// TIA Portal V17 export
// export: Created 2025-03-07T09:19:56.0957426Z, ExportSetting WithDefaults, DisplayName Totally Integrated Automation Portal, DisplayVersion V17 Update 8, DisplayName TIA Portal Openness, DisplayVersion V17 Update 8, DisplayName TIA Portal Version Control Interface, DisplayVersion V17, DisplayName SINAMICS Startdrive Advanced, DisplayVersion V17 SP2, DisplayName SINAMICS Startdrive G110M, G120, G120C, G120D, G120P, G115D, DisplayVersion V17 SP2, DisplayName SINAMICS Startdrive G130, G150, S120, S150, SINAMICS MV, S210, DisplayVersion V17 SP2, DisplayName STEP 7 Professional, DisplayVersion V17 Update 8, DisplayName SINUMERIK ONE STEP 7 Toolbox, DisplayVersion V17 Update 12, DisplayName SINUMERIK 840D sl STEP 7 Toolbox, DisplayVersion V17 Update 12, DisplayName STEP 7 Safety, DisplayVersion V17 Update 6, DisplayName WinCC Advanced, DisplayVersion V17 Update 8
TYPE "LOAD_ROBOT"
// stored: IsFailsafeCompliant false
   STRUCT
      TO_FIXT : Struct
         PART_A_LOADED_FIXT1 : Bool;   // PART 1 LOADED ARM 1 / PART A LOADED FIXT 1
         PART_B_LOADED_FIXT1 : Bool;   // PART 2 LOADED ARM 1 / PART B LOADED FIXT 1
         PART_C_LOADED_FIXT1 : Bool;   // PART 3 LOADED ARM 1 / PART C LOADED FIXT 1
         PART_D_LOADED_FIXT1 : Bool;   // PART 4 LOADED ARM 1 / PART D LOADED FIXT 1
         PART_A_LOADED_FIXT2 : Bool;   // PART 1 LOADED ARM 2 / PART A LOADED FIXT 2
         PART_B_LOADED_FIXT2 : Bool;   // PART 2 LOADED ARM 2 / PART B LOADED FIXT 2
         PART_C_LOADED_FIXT2 : Bool;   // PART 3 LOADED ARM 2 / PART C LOADED FIXT 2
         PART_D_LOADED_FIXT2 : Bool;   // PART 4 LOADED ARM 2 / PART D LOADED FIXT 2
         PARTS_LOADED_FIXT1 : Bool;   // PARTS LOADED ARM 1 / PARTS LOADED FIXT 1
         PARTS_LOADED_FIXT2 : Bool;   // PARTS LOADED ARM 2 / PARTS LOADED FIXT 2
         I_PART_PRESENT_A : Bool;   // INPUT PART PRESENT A
         I_PART_PRESENT_B : Bool;   // INPUT PART PRESENT B
         I_PART_PRESENT_C : Bool;   // INPUT PART PRESENT C
         I_PART_PRESENT_D : Bool;   // INPUT PART PRESENT D
         PART_A_UNLOADED_FIXT1 : Bool;   // PART 1 UNLOADED ARM 1 / PART A UNLOADED FIXT 1
         PART_B_UNLOADED_FIXT1 : Bool;   // PART 2 UNLOADED ARM 1 / PART B UNLOADED FIXT 1
         PART_C_UNLOADED_FIXT1 : Bool;   // PART 3 UNLOADED ARM 1 / PART C UNLOADED FIXT 1
         PART_D_UNLOADED_FIXT1 : Bool;   // PART 4 UNLOADED ARM 1 / PART D UNLOADED FIXT 1
         PART_A_UNLOADED_FIXT2 : Bool;   // PART 1 UNLOADED ARM 2 / PART A UNLOADED FIXT 2
         PART_B_UNLOADED_FIXT2 : Bool;   // PART 2 UNLOADED ARM 2 / PART B UNLOADED FIXT 2
         PART_C_UNLOADED_FIXT2 : Bool;   // PART 3 UNLOADED ARM 2 / PART C UNLOADED FIXT 2
         PART_D_UNLOADED_FIXT2 : Bool;   // PART 4 UNLOADED ARM 2 / PART D UNLOADED FIXT 2
         PARTS_UNLOADED_FIXT1 : Bool;   // PARTS UNLOADED ARM 1 / PARTS UNLOADED FIXT 1
         PARTS_UNLOADED_FIXT2 : Bool;   // PARTS UNLOADED ARM 2 / PARTS UNLOADED FIXT 2
         AUX_PART_A_LOADED_FIXT1 : Bool;   // AUX PART A LOADED FIXT1
         AUX_PART_B_LOADED_FIXT1 : Bool;   // AUX PART B LOADED FIXT1
         AUX_PART_C_LOADED_FIXT1 : Bool;   // AUX PART C LOADED FIXT1
         AUX_PART_D_LOADED_FIXT1 : Bool;   // AUX PART D LOADED FIXT1
         AUX_PART_A_LOADED_FIXT2 : Bool;   // AUX PART A LOADED FIXT2
         AUX_PART_B_LOADED_FIXT2 : Bool;   // AUX PART B LOADED FIXT2
         AUX_PART_C_LOADED_FIXT2 : Bool;   // AUX PART C LOADED FIXT2
         AUX_PART_D_LOADED_FIXT2 : Bool;   // AUX PART D LOADED FIXT2
         NO_PARTS_AT_FIXT1 : Bool;   // NO PARTS AT ARM 1 / NO PARTS AT FIXT 1
         NO_PARTS_AT_FIXT2 : Bool;   // NO PARTS AT ARM 2 / NO PARTS AT FIXT 2
         PART_A_LOADED_FIXT1_P : Bool;   // PART 1 LOADED ARM 1 PULSE / PART A LOADED FIXT 1 PULSE
         PART_B_LOADED_FIXT1_P : Bool;   // PART 2 LOADED ARM 1 PULSE / PART B LOADED FIXT 1 PULSE
         PART_C_LOADED_FIXT1_P : Bool;   // PART 3 LOADED ARM 1 PULSE / PART C LOADED FIXT 1 PULSE
         PART_D_LOADED_FIXT1_P : Bool;   // PART 4 LOADED ARM 1 PULSE / PART D LOADED FIXT 1 PULSE
         PART_A_LOADED_FIXT2_P : Bool;   // PART 1 LOADED ARM 2 PULSE / PART A LOADED FIXT 2 PULSE
         PART_B_LOADED_FIXT2_P : Bool;   // PART 2 LOADED ARM 2 PULSE / PART B LOADED FIXT 2 PULSE
         PART_C_LOADED_FIXT2_P : Bool;   // PART 3 LOADED ARM 2 PULSE / PART C LOADED FIXT 2 PULSE
         PART_D_LOADED_FIXT2_P : Bool;   // PART 4 LOADED ARM 2 PULSE / PART D LOADED FIXT 2 PULSE
         PARTS_LOADED_FIXT1_P : Bool;   // PARTS LOADED ARM 1 PULSE / PARTS LOADED FIXT 1 PULSE
         PARTS_LOADED_FIXT2_P : Bool;   // PARTS LOADED ARM 2 PULSE / PARTS LOADED FIXT 2 PULSE
         ANY_PART_LOADED : Bool;   // ANY PART LOADED
         ANY_PART_UNLOADED : Bool;   // ANY PART UNLOADED
         ENABLE_LOAD_UNLOAD : Bool;   // ENABLE TO LOAD UNLOAD LOADER TO TRANSFER
         PARTS_LOADING : Bool;   // THE GANTRY IS LOADING PARTS
         PART_A_UNLOADED_FIXT1_P : Bool;   // PART 1 UNLOADED ARM 1 PULSE / PART A UNLOADED FIXT 1 PULSE
         PART_B_UNLOADED_FIXT1_P : Bool;   // PART 2 UNLOADED ARM 1 PULSE / PART B UNLOADED FIXT 1 PULSE
         PART_C_UNLOADED_FIXT1_P : Bool;   // PART 3 UNLOADED ARM 1 PULSE / PART C UNLOADED FIXT 1 PULSE
         PART_D_UNLOADED_FIXT1_P : Bool;   // PART 4 UNLOADED ARM 1 PULSE / PART D UNLOADED FIXT 1 PULSE
         PART_A_UNLOADED_FIXT2_P : Bool;   // PART 1 UNLOADED ARM 2 PULSE / PART A UNLOADED FIXT 2 PULSE
         PART_B_UNLOADED_FIXT2_P : Bool;   // PART 2 UNLOADED ARM 2 PULSE / PART B UNLOADED FIXT 2 PULSE
         PART_C_UNLOADED_FIXT2_P : Bool;   // PART 3 UNLOADED ARM 2 PULSE / PART C UNLOADED FIXT 2 PULSE
         PART_D_UNLOADED_FIXT2_P : Bool;   // PART 4 UNLOADED ARM 2 PULSE / PART D UNLOADED FIXT 2 PULSE
         PARTS_UNLOADED_FIXT1_P : Bool;   // PARTS UNLOADED ARM 1 PULSE / PARTS UNLOADED FIXT 1 PULSE
         PARTS_UNLOADED_FIXT2_P : Bool;   // PARTS UNLOADED ARM 2 PULSE / PARTS UNLOADED FIXT 2 PULSE
         PARTS_UNLOADING : Bool;   // THE GANTRY IS UNLOADING PARTS
         ACK_REJECT_PART_A_FX2 : Bool;   // ACKNOWLEDGE REJECT PART A FROM FIXTURE 2
         ACK_REJECT_PART_B_FX2 : Bool;   // ACKNOWLEDGE REJECT PART B FROM FIXTURE 2
         ACK_REJECT_PART_C_FX2 : Bool;   // ACKNOWLEDGE REJECT PART C FROM FIXTURE 2
         ACK_REJECT_PART_D_FX2 : Bool;   // ACKNOWLEDGE REJECT PART D FROM FIXTURE 2
      END_STRUCT;
      FROM_FIXT : Struct
         REQ_LOAD_PART_A_FIXT1 : Bool;   // REQUEST LOAD PART 1 ARM 1 / REQUEST LOAD PART A FIXT 1
         REQ_LOAD_PART_B_FIXT1 : Bool;   // REQUEST LOAD PART 2 ARM 1 / REQUEST LOAD PART B FIXT 1
         REQ_LOAD_PART_C_FIXT1 : Bool;   // REQUEST LOAD PART 3 ARM 1 / REQUEST LOAD PART C FIXT 1
         REQ_LOAD_PART_D_FIXT1 : Bool;   // REQUEST LOAD PART 4 ARM 1 / REQUEST LOAD PART D FIXT 1
         REQ_LOAD_PART_A_FIXT2 : Bool;   // REQUEST LOAD PART 1 ARM 2 / REQUEST LOAD PART A FIXT 2
         REQ_LOAD_PART_B_FIXT2 : Bool;   // REQUEST LOAD PART 2 ARM 2 / REQUEST LOAD PART B FIXT 2
         REQ_LOAD_PART_C_FIXT2 : Bool;   // REQUEST LOAD PART 3 ARM 2 / REQUEST LOAD PART C FIXT 2
         REQ_LOAD_PART_D_FIXT2 : Bool;   // REQUEST LOAD PART 4 ARM 2 / REQUEST LOAD PART D FIXT 2
         REQUEST_LOAD_PARTS : Bool;   // REQUEST LOAD PARTS
         REQ_UNLOAD_PART_A_FIXT1 : Bool;   // REQUEST UNLOAD PART 1 ARM 1 / REQUEST UNLOAD PART A FIXT 1
         REQ_UNLOAD_PART_B_FIXT1 : Bool;   // REQUEST UNLOAD PART 2 ARM 1 / REQUEST UNLOAD PART B FIXT 1
         REQ_UNLOAD_PART_C_FIXT1 : Bool;   // REQUEST UNLOAD PART 3 ARM 1 / REQUEST UNLOAD PART C FIXT 1
         REQ_UNLOAD_PART_D_FIXT1 : Bool;   // REQUEST UNLOAD PART 4 ARM 1 / REQUEST UNLOAD PART D FIXT 1
         REQ_UNLOAD_PART_A_FIXT2 : Bool;   // REQUEST UNLOAD PART 1 ARM 2 / REQUEST UNLOAD PART A FIXT 2
         REQ_UNLOAD_PART_B_FIXT2 : Bool;   // REQUEST UNLOAD PART 2 ARM 2 / REQUEST UNLOAD PART B FIXT 2
         REQ_UNLOAD_PART_C_FIXT2 : Bool;   // REQUEST UNLOAD PART 3 ARM 2 / REQUEST UNLOAD PART C FIXT 2
         REQ_UNLOAD_PART_D_FIXT2 : Bool;   // REQUEST UNLOAD PART 4 ARM 2 / REQUEST UNLOAD PART D FIXT 2
         REQUEST_UNLOAD_PARTS : Bool;   // REQUEST UNLOAD PARTS
         PART_ID : Byte;   // PART ID
         NEST_FIXTURE : Byte;   // NEST FIXTURE
         PART_TYPE : Byte;   // PART TYPE
         PART_TYPE_NEST_UNLD : Byte;   // PART TYPE NEST UNLOAD
         BYTE8 : Byte;
         BYTE9 : Byte;
         BYTE10 : Byte;
         MACHINE_READY_FOR_OPERAT : Bool;   // MACHINED READY FOR OPERATION
      END_STRUCT;
   END_STRUCT;
END_TYPE
